    movel([0.236549, -1.049245, -2.641806, -1.021338, 1.570796, 1.807346],accel_mss,speed_ms,0,blend_radius_m)
    movel([0.236549, -1.047583, -2.640504, -1.024302, 1.570796, 1.807346],accel_mss,speed_ms,0,blend_radius_m)
    movel([0.236549, -1.045934, -2.639200, -1.027256, 1.570796, 1.807346],accel_mss,speed_ms,0,blend_radius_m)
    movel([0.236549, -1.044296, -2.637893, -1.030200, 1.570796, 1.807346],accel_mss,speed_ms,0,blend_radius_m)
    movel([0.236549, -1.042670, -2.636585, -1.033134, 1.570796, 1.807346],accel_mss,speed_ms,0,blend_radius_m)
    movel([0.236549, -1.041056, -2.635274, -1.036059, 1.570796, 1.807346],accel_mss,speed_ms,0,blend_radius_m)
    movel([0.236549, -1.039454, -2.633962, -1.038974, 1.570796, 1.807346],accel_mss,speed_ms,0,blend_radius_m)
    movel([0.236549, -1.037863, -2.632647, -1.041879, 1.570796, 1.807346],accel_mss,speed_ms,0,blend_radius_m)
    # End of main program
  end

  Machining1()
end
